FUNCTION_BLOCK xPPU_Crane
VAR_INPUT
	i_error: POINTER TO ErrorManager;
	i_process: POINTER TO ProcessManager;
	i_state: POINTER TO StateTracker;
END_VAR
VAR
	m_emptyParams: ParameterSet;
	m_subRes: EOperationResult;
END_VAR

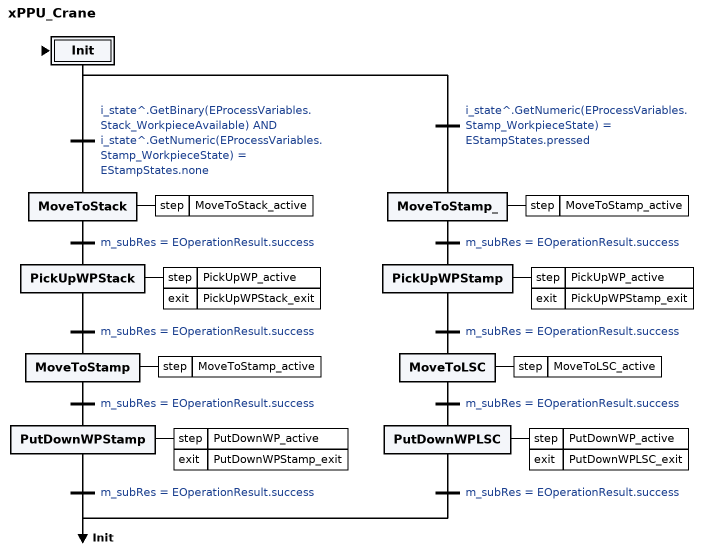
INITIAL_STEP Init:
END_STEP
TRANSITION FROM Init TO MoveToStack
    := i_state^.GetBinary(EProcessVariables.Stack_WorkpieceAvailable) AND i_state^.GetNumeric(EProcessVariables.Stamp_WorkpieceState) = EStampStates.none;
END_TRANSITION
STEP MoveToStack:
    MoveToStack_active(N);  // step action
END_STEP
TRANSITION FROM MoveToStack TO PickUpWPStack
    := m_subRes = EOperationResult.success;
END_TRANSITION
STEP PickUpWPStack:
    PickUpWP_active(N);  // step action
    PickUpWPStack_exit(P0);  // exit action
END_STEP
TRANSITION FROM PickUpWPStack TO MoveToStamp
    := m_subRes = EOperationResult.success;
END_TRANSITION
STEP MoveToStamp:
    MoveToStamp_active(N);  // step action
END_STEP
TRANSITION FROM MoveToStamp TO PutDownWPStamp
    := m_subRes = EOperationResult.success;
END_TRANSITION
STEP PutDownWPStamp:
    PutDownWP_active(N);  // step action
    PutDownWPStamp_exit(P0);  // exit action
END_STEP
TRANSITION FROM PutDownWPStamp TO Init
    := m_subRes = EOperationResult.success;
END_TRANSITION
TRANSITION FROM Init TO MoveToStamp_
    := i_state^.GetNumeric(EProcessVariables.Stamp_WorkpieceState) = EStampStates.pressed;
END_TRANSITION
STEP MoveToStamp_:
    MoveToStamp_active(N);  // step action
END_STEP
TRANSITION FROM MoveToStamp_ TO PickUpWPStamp
    := m_subRes = EOperationResult.success;
END_TRANSITION
STEP PickUpWPStamp:
    PickUpWP_active(N);  // step action
    PickUpWPStamp_exit(P0);  // exit action
END_STEP
TRANSITION FROM PickUpWPStamp TO MoveToLSC
    := m_subRes = EOperationResult.success;
END_TRANSITION
STEP MoveToLSC:
    MoveToLSC_active(N);  // step action
END_STEP
TRANSITION FROM MoveToLSC TO PutDownWPLSC
    := m_subRes = EOperationResult.success;
END_TRANSITION
STEP PutDownWPLSC:
    PutDownWP_active(N);  // step action
    PutDownWPLSC_exit(P0);  // exit action
END_STEP
TRANSITION FROM PutDownWPLSC TO Init
    := m_subRes = EOperationResult.success;
END_TRANSITION

ACTION MoveToLSC_active:
m_subRes := i_process^.Execute(
	EBehaviorType.control_primitive,
	EPrimitives.Crane_MoveToLSC,
	m_emptyParams);
END_ACTION

ACTION MoveToStack_active:
m_subRes := i_process^.Execute(
	EBehaviorType.control_primitive,
	EPrimitives.Crane_MoveToStack,
	m_emptyParams);
END_ACTION

ACTION MoveToStamp_active:
m_subRes := i_process^.Execute(
	EBehaviorType.control_primitive,
	EPrimitives.Crane_MoveToStamp,
	m_emptyParams);
END_ACTION

ACTION PickUpWP_active:
m_subRes := i_process^.Execute(
	EBehaviorType.control_primitive,
	EPrimitives.Crane_PickUpWP,
	m_emptyParams);
END_ACTION

ACTION PickUpWPStack_exit:
i_state^.ShiftProduct(EProducts.stack_product, EProducts.crane_product);
END_ACTION

ACTION PickUpWPStamp_exit:
i_state^.ShiftProduct(EProducts.stamp_product, EProducts.crane_product);
END_ACTION

ACTION PutDownWP_active:
m_subRes := i_process^.Execute(
	EBehaviorType.control_primitive,
	EPrimitives.Crane_PutDownWP,
	m_emptyParams);
END_ACTION

ACTION PutDownWPLSC_exit:
i_state^.ShiftProduct(EProducts.crane_product, EProducts.LSC_product);
END_ACTION

ACTION PutDownWPStamp_exit:
i_state^.ShiftProduct(EProducts.crane_product, EProducts.stamp_product);
END_ACTION

END_FUNCTION_BLOCK

(* stored: Version 1.1.0.1, ProductVersion 3.1.4024.12
   POU xPPU_Crane: Id {78161606-71b4-4291-9ac3-095c552c2798}, SpecialFunc None
   Action MoveToLSC_active: Id {8277d77e-cd34-4ec5-9f75-b93467ba1bb6}
   Action MoveToStack_active: Id {571b406f-6c8e-4544-9ae9-49953b6b39be}
   Action MoveToStamp_active: Id {a7848926-ee25-41bb-a037-2f10498f3c62}
   Action PickUpWP_active: Id {0442f4fd-88ed-4177-bc1f-6efb591dfd4d}
   Action PickUpWPStack_exit: Id {1b736f68-d7a0-4bc6-af85-9b732ac83761}
   Action PickUpWPStamp_exit: Id {6d99610e-69d1-409d-88f0-202e27f184fb}
   Action PutDownWP_active: Id {c713f15e-67e6-4a12-b1c1-93deb7666c90}
   Action PutDownWPLSC_exit: Id {f398bd84-d715-4628-8579-139e0657ea82}
   Action PutDownWPStamp_exit: Id {39d022ad-1212-45a5-b9d2-c0ff009b69d4} *)
